// Removes outdated messages from the buffer
FUNCTION F_Remove : BOOL
VAR_INPUT
END_VAR
VAR
    nIndex:					UDINT;
END_VAR
(*
    Tc3_Event – TwinCAT 3 Event Logging Framework
    Copyright (c) Peter Zerlauth

    This component is provided under a Dual Licensing Model:

    1. GPLv3 Open-Source License
       - Free for personal, educational, and non-commercial use.
       - Commercial use allowed only if the entire application is published
         under GPLv3, including all modifications to this code.
       - Requires full disclosure of source code for derivative works.

    2. Commercial License
       - Required for integration into proprietary or closed-source products.
       - Removes all GPLv3 copyleft obligations.
       - Includes optional warranty, professional support, and long-term
         maintenance options.

    For commercial licensing, contact:
        info@peterzerlauth.com

    By using this Function Block you agree to the terms of the selected license.
*)

// just once a cycle
IF GVL.nFunction <> GVL.nTimestamp THEN
	GVL.nFunction:= GVL.nTimestamp;
	// Remove outdated messages
	WHILE nIndex < GVL.nBuffer DO
		IF (GVL.nTimestamp - GVL.aBuffer[nIndex].nTimestamp) > 1_000_000_000 THEN // 1 s = 1e9 ns
			// Shift remaining messages down
			MEMMOVE(ADR(GVL.aBuffer[nIndex]), ADR(GVL.aBuffer[nIndex + 1]), SIZEOF(FB_Message) * (GVL.nBuffer - nIndex - 1));
			GVL.nBuffer := GVL.nBuffer - 1;
			F_Remove := TRUE;
		ELSE
			nIndex := nIndex + 1;
		END_IF
	END_WHILE
END_IF

END_FUNCTION

(* stored: Version 1.1.0.1
   POU F_Remove: Id {d773492b-347d-47bd-87c4-88c07813c65f}, SpecialFunc None *)
